DATA_BLOCK "LCC_ConfigDevice_DB"
{ S7_Optimized_Access := 'TRUE' }
AUTHOR : SIOS
FAMILY : LCC
VERSION : 1.0
NON_RETAIN
"LCC_ConfigDevice"

BEGIN

END_DATA_BLOCK

